FUNCTION CheckDivReal : REAL
VAR_INPUT
    divisor : REAL;
END_VAR
VAR
END_VAR

IF divisor = 0 THEN
    CheckDivReal := 1;
ELSE
    CheckDivReal := divisor;
END_IF

END_FUNCTION

(* stored: Version 1.1.0.1, ProductVersion 3.1.4024.12
   POU CheckDivReal: Id {1da362bf-0e78-4cea-a6d9-6183f9f81351}, SpecialFunc None *)
